{attribute 'qualified_only'}
VAR_GLOBAL PERSISTENT 
	Lot: LotDataType;
END_VAR

(* stored: Version 1.1.0.1, ProductVersion 3.1.4020.12
   GVL LotsData: Id {a61e95d1-c161-4d97-81ba-36f31af0c433} *)
